// TIA Portal V20 export
ORGANIZATION_BLOCK "Pull or plug of modules"   // OB83, FBD, PullOrPlugOfModules
{ S7_Optimized_Access := 'TRUE' }
// stored: SetENOAutomatically false
   VAR_INPUT
      LADDR : HW_IO;   // Hardware identifier
      Event_Class : Byte;   // 16#38/39: module inserted, removed
      Fault_ID : Byte;   // Fault identifier
   END_VAR
BEGIN

NETWORK
TITLE = call diagnose
      CALL  "Diag", "Diag_DB";

END_ORGANIZATION_BLOCK
